(*

.. <legal notes>

legal notes
=================
| SPDX-FileCopyrightText: © 2026 Oleksandr Tiutyk <trofimich@gmail.com>
| SPDX-License-Identifier: LGPL-3.0-only
| For details check: LGPL-3.0-only_

.. _LGPL-3.0-only: https://www.gnu.org/licenses/lgpl-3.0.en.html

.. </legal notes>

*)

PROGRAM UsignedInt32Helper
VAR CONSTANT
	MIN_VALUE : UDINT := 0;
	MAX_VALUE : UDINT := 4_294_967_295;
END_VAR
VAR
	_ClassName : STRING := __POUNAME();
END_VAR

{attribute 'monitoring' := 'call'}
PROPERTY ClassName : STRING
GET
ClassName := _ClassName;
END_GET
END_PROPERTY

{attribute 'monitoring' := 'call'}
PROPERTY NamespaceName : STRING
GET
NamespaceName := CurrentNamespace.Name;
END_GET
END_PROPERTY

END_PROGRAM

(* stored: Version 1.1.0.1
   POU UsignedInt32Helper: Id {6bac338b-229a-43e9-a30f-455531e1f310}, SpecialFunc None
   Property ClassName: Id {078f51d7-7a9e-4bef-a7f8-cb5013aa458a}
   Get Get: Id {c0ad2f36-6652-4fd6-8323-ef857fb2ba2a}
   Property NamespaceName: Id {ee80b6e7-69cd-4ea9-a37e-1cd7459c76b6}
   Get Get: Id {e83e0b93-d2f7-4e66-89bd-17343024db2f} *)
